// TIA Portal V20 export
DATA_BLOCK "Config"   // DB47
// stored: MemoryReserve 100, Namespace Unit1.Em6
   VAR
      em : "LAF_typeEmConfiguration";   // Configuration of EM Parameters
      cmHotpressLeftSafetyPin : "LBC_typeDigitalSignalConfiguration";
      cmHotpressLeftJRDetect : "LBC_typeDigitalSignalConfiguration";
      cmHotpressLeftStageLiftFrontUpDown : "LBC_typeTwoWayActuatorConfiguration";
      cmHotpressLeftStageLiftRearUpDown : "LBC_typeTwoWayActuatorConfiguration";
      cmHotpressLeftStageLiftAllUpDown : "LBC_typeTwoWayActuatorConfiguration";
      cmHotPressLeftServoPress : "LER_typeServoPressConfiguration";
      cmHotPressLeftTemperature : "LER_typeHeaterConfiguration";
   END_VAR
BEGIN
   em.referenceDesignator.parent := WSTRING#'U1';
   em.referenceDesignator.relative := WSTRING#'EM0';
   cmHotpressLeftStageLiftFrontUpDown.referenceDesignator := WSTRING#'STAGE LIFT';
   cmHotpressLeftStageLiftFrontUpDown.monitoringDiscrepancy := T#5s;
   cmHotpressLeftStageLiftRearUpDown.referenceDesignator := WSTRING#'STAGE LIFT';
   cmHotpressLeftStageLiftRearUpDown.monitoringDiscrepancy := T#5s;
   cmHotpressLeftStageLiftAllUpDown.referenceDesignator := WSTRING#'STAGE LIFT';
   cmHotpressLeftStageLiftAllUpDown.monitoringDiscrepancy := T#5s;
   cmHotPressLeftServoPress.hwID."220ByteIn" := 621;
   cmHotPressLeftServoPress.hwID."220ByteOut" := 622;
   cmHotPressLeftTemperature.MB_Comm_Load.PORT := 1055;
   cmHotPressLeftTemperature.MB_Comm_Load.BAUD := 9600;
   cmHotPressLeftTemperature.MB_Comm_Load.PARITY := 2;
END_DATA_BLOCK
